FUNCTION_BLOCK FB_Pusher
VAR_INPUT
	SENSOR : BOOL;
	FRONTAL	: BOOL;
	CAMARA: BOOL;
END_VAR
VAR_OUTPUT
	PUSHER : BOOL;
END_VAR
VAR
	FTRIGA : F_TRIG;
END_VAR

FTRIGA(CLK:= SENSOR);

IF CAMARA AND FTRIGA.Q THEN
	PUSHER := TRUE;	 
END_IF

IF FRONTAL THEN
	PUSHER := FALSE;
END_IF

END_FUNCTION_BLOCK

(* stored: Version 1.1.0.1, ProductVersion 3.1.4024.12
   POU FB_Pusher: Id {303d9187-b056-437c-b760-a6cbeaa7a0c4}, SpecialFunc None *)
